{attribute 'qualified_only'}
{attribute 'strict'}
{attribute 'to_string'}
TYPE ePSBMode :
(
	None 				:= 0,
	Monitor				:= 1,
	MonitorControl		:= 2	
);
END_TYPE

(* stored: Version 1.1.0.1, ProductVersion 3.1.4026.18
   DUT ePSBMode: Id {b4d662ec-6b70-44e5-bdab-328e228429f1} *)
